FUNCTION_BLOCK FB_CtrlgxParser
VAR_INPUT
END_VAR
VAR_OUTPUT
END_VAR
VAR
END_VAR
xdfsdfsd

END_FUNCTION_BLOCK

(* stored: Version 1.1.0.1, ProductVersion 3.1.4022.12
   POU FB_CtrlgxParser: Id {dd46f8b2-f737-4b53-be6c-229c4eef03e8}, SpecialFunc None *)
